FUNCTION_BLOCK FB_Http_Client
VAR_INPUT
	i_bExecute 			: BOOL;
	i_sAmsNetId			: STRING;
	i_stHttpRequest 	: ST_HTTP_Request;
	i_sRemoteHost		: STRING(255);
END_VAR
VAR_OUTPUT	
	o_bBusy				: BOOL;
	o_bError			: BOOL;
	o_udErrorId			: UDINT;
	o_sErrorTxt			: STRING;
	o_bDataReceived		: BOOL;	
	o_stHttpResponse	: ST_HTTP_Response;
END_VAR
VAR
	fbGetHttpConnectionParams: FB_GetHttpConnectionParams;
	fbSocketConnect		: FB_SocketConnect;
	fbSocketSend		: FB_SocketSend;
	fbSocketReceive		: FB_SocketReceive;
	fbSocketClose		: FB_SocketClose;
	bGetHttpConnectionParams: BOOL;
	bSocketConnect		: BOOL;
	bSocketSend			: BOOL;
	bSocketReceive		: BOOL;
	bSocketClose		: BOOL;
	nState				: INT := 10;
	hSocket				: T_HSOCKET;
	udBytesToSend		: UDINT;
	arrBytesToSend		: ARRAY[0..HTTP_SEND_DATA_ARRAY_SIZE] OF BYTE;
	tTimeOut			: TIME := T#10S;
	arrReceivedBytes	: ARRAY[0..HTTP_RECEIVE_DATA_ARRAY_SIZE] OF BYTE;
	bHttpConnParamsParamsParsed : BOOL;
	stHttpConnectionParams : ST_HTTP_Connection_Parameters;
	udReceivedBytes		: UDINT;
	Delay_TON			: TON;
END_VAR



CASE nState OF

10: (* Initial state *)
	nState := 20;
	
20:	(* Waiting for start *)

	IF i_bExecute THEN
		
		MEMSET(ADR(arrReceivedBytes), 0, SIZEOF(arrReceivedBytes));
		o_bDataReceived := FALSE;
		udReceivedBytes := 0;
		o_udErrorId		:= 0;
		o_bError 		:= FALSE;
		o_sErrorTxt 	:= '';
		o_bBusy 		:= TRUE;
		
		IF NOT bHttpConnParamsParamsParsed THEN
			bGetHttpConnectionParams := TRUE;
			nState := 25;
		ELSE
			bSocketConnect 	:= TRUE;
			nState 			:= 30;
		END_IF
		
	END_IF

25:	(* Waiting for addr resolved *)


	IF fbGetHttpConnectionParams.o_bError THEN
		o_udErrorId := fbGetHttpConnectionParams.o_nErrId;
		o_sErrorTxt := 'FB_GetHttpConnectionParams error';
		nState 		:= 100; 
	ELSIF fbGetHttpConnectionParams.o_bReady THEN
		stHttpConnectionParams := fbGetHttpConnectionParams.o_stHttpConnectionParams;
		bHttpConnParamsParamsParsed := TRUE;
		bSocketConnect 	:= TRUE;
		nState 			:= 30;
	END_IF	

30:	(* Waiting for connect *)

	IF fbSocketConnect.bError THEN
		o_udErrorId := fbSocketConnect.nErrId;
		o_sErrorTxt := 'FB_SocketConnect error';
		nState 		:= 100; 
	ELSIF NOT fbSocketConnect.bBusy THEN
		
		CASE i_stHttpRequest.eHttpRequestType OF 
			
			E_HTTP_Request_Type_GET:			
					udBytesToSend 	:= F_BuildHttpGetRequest(ADR(i_stHttpRequest), stHttpConnectionParams, arrBytesToSend);
							
			E_HTTP_Request_Type_POST:			
					udBytesToSend 	:= F_BuildHttpPostRequest(ADR(i_stHttpRequest), stHttpConnectionParams, arrBytesToSend);
							
		END_CASE

		bSocketSend		:= TRUE;
		nState 			:= 40; 		
	END_IF

40:	(* Waiting for send *) 

	IF fbSocketSend.bError THEN
		o_udErrorId := fbSocketSend.nErrId;
		o_sErrorTxt := 'FB_SocketSend error';
		nState 		:= 100; 
	ELSIF NOT fbSocketSend.bBusy THEN
		bSocketReceive	:= TRUE;
		nState 			:= 50; 		
	END_IF
	
50:	(* Waiting for receive *)

	// Timeout
	Delay_TON(IN := TRUE, PT := T#1500MS);
	
	IF fbSocketReceive.bError THEN
		Delay_TON(IN := FALSE);
		o_udErrorId := fbSocketReceive.nErrId;
		o_sErrorTxt := 'FB_SocketReceive error';
		nState 		:= 100; 
	ELSIF NOT fbSocketReceive.bBusy THEN
		IF fbSocketReceive.nRecBytes > 0 THEN
			Delay_TON(IN := FALSE);
			o_bDataReceived := TRUE;
			udReceivedBytes := fbSocketReceive.nRecBytes;
			o_stHttpResponse:= F_ParseHttpResponse(i_udNumOfBytes := udReceivedBytes, io_arrReceivedBytes:= arrReceivedBytes);
			bSocketClose	:= TRUE;
			nState 			:= 60;
		ELSIF Delay_TON.Q THEN
			Delay_TON(IN := FALSE);
			bSocketClose	:= TRUE;
			nState 			:= 60;
		ELSE
			bSocketReceive	:= TRUE;
		END_IF
	END_IF

60:	(* Waiting for close *)

	IF fbSocketClose.bError THEN
		o_udErrorId := fbSocketClose.nErrId;
		o_sErrorTxt := 'FB_SocketReceive error';
		nState 		:= 100; 
	ELSIF NOT fbSocketClose.bBusy THEN
		nState 	:= 10; 		
		o_bBusy := FALSE;
	END_IF

100:	(* Error *)

	o_bBusy  := FALSE;
	o_bError := TRUE;
	IF NOT i_bExecute THEN
		nState := 10;
	END_IF

END_CASE

ACT_FB_Calls();

bGetHttpConnectionParams := FALSE;
bSocketConnect 	:= FALSE;
bSocketSend 	:= FALSE;
bSocketReceive 	:= FALSE;
bSocketClose 	:= FALSE;

ACTION ACT_FB_Calls:
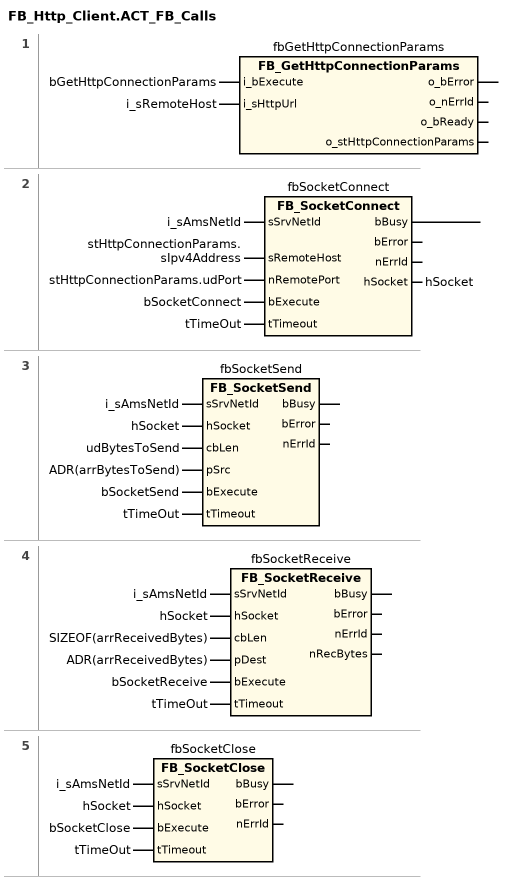
// NETWORK 1
fbGetHttpConnectionParams(i_bExecute := bGetHttpConnectionParams, i_sHttpUrl := i_sRemoteHost); // FB_GetHttpConnectionParams

// NETWORK 2
fbSocketConnect(
    sSrvNetId := i_sAmsNetId,
    sRemoteHost := stHttpConnectionParams.sIpv4Address,
    nRemotePort := stHttpConnectionParams.udPort,
    bExecute := bSocketConnect,
    tTimeout := tTimeOut,
    hSocket => hSocket); // FB_SocketConnect

// NETWORK 3
fbSocketSend(
    sSrvNetId := i_sAmsNetId,
    hSocket := hSocket,
    cbLen := udBytesToSend,
    pSrc := ADR(arrBytesToSend),
    bExecute := bSocketSend,
    tTimeout := tTimeOut); // FB_SocketSend

// NETWORK 4
fbSocketReceive(
    sSrvNetId := i_sAmsNetId,
    hSocket := hSocket,
    cbLen := SIZEOF(arrReceivedBytes),
    pDest := ADR(arrReceivedBytes),
    bExecute := bSocketReceive,
    tTimeout := tTimeOut); // FB_SocketReceive

// NETWORK 5
fbSocketClose(sSrvNetId := i_sAmsNetId, hSocket := hSocket, bExecute := bSocketClose, tTimeout := tTimeOut); // FB_SocketClose
END_ACTION

END_FUNCTION_BLOCK

(* stored: Version 1.1.0.1, ProductVersion 3.1.4020.12
   POU FB_Http_Client: Id {68e62783-2ed7-4de8-a59e-37c698a3a109}, SpecialFunc None
   Action ACT_FB_Calls: Id {7aaaca00-f5c3-474b-97f4-753cceeca101} *)
